Fanuc KAREL source: kb00018.KL

-- PROVISIONAL review KL for V770-1; original PC SHA256 7889453acdedd942db2f3b5823a36902b9c0a98d604895fe8f356b8ec6220c98
-- Incomplete behavior may be omitted. Consult companion uncertainty JSON. Do not deploy.
PROGRAM KB00018
%NOLOCKGROUP
BEGIN
  -- UNRESOLVED_PC offsets 5-12; opcodes 9D,23
  -- UNRESOLVED_PC offsets 17-65; opcodes 27,22,1C,22,1C,22,1C,22,27,9D,31
  -- UNRESOLVED_PC offsets 70-74; opcodes 7F
END KB00018
